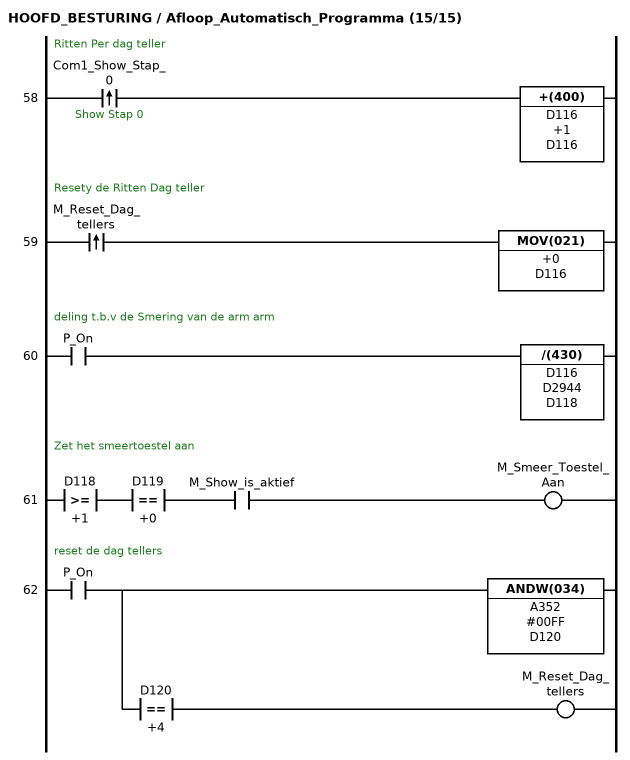
; [picture p120: HOOFD_BESTURING / Afloop_Automatisch_Programma, rungs 58-62]
; rung 58: Ritten Per dag teller
@LD Com1_Show_Stap_0  ; Show Stap 0
+(400) D116 +1 D116
; rung 59: Resety de Ritten Dag teller
@LD M_Reset_Dag_tellers
MOV(021) +0 D116
; rung 60: deling t.b.v de Smering van de arm arm
LD P_On
/(430) D116 D2944 D118
; rung 61: Zet het smeertoestel aan
LD>=S(327) D118 +1
AND=S(302) D119 +0
AND M_Show_is_aktief
OUT M_Smeer_Toestel_Aan
; rung 62: reset de dag tellers
LD P_On
ANDW(034) A352 #00FF D120
AND=S(302) D120 +4
OUT M_Reset_Dag_tellers

### Section Einde_Hoofd_Besturing
; rung 0
END(001)

## Program SIGNALEN_GROND (cyclic task 5)
Local symbols
D_FACTOR_01 D5132 REAL  ; DIVERTION FACTOR IN REAL FORMAT
D_HELP2_CNT2 D5140 REAL  ; RESULT AFTER MULIPLYING IN REAL FORMAT
D_HELP3_CNT1 D5134 REAL  ; RESULT AFTER DIVERTING IN REAL FORMAT
D_HELP3_CNT2 D5144 REAL  ; RESULT AFTER DIVERTING IN REAL FORMAT

### Section Incremental_Encoder_Decoder_1

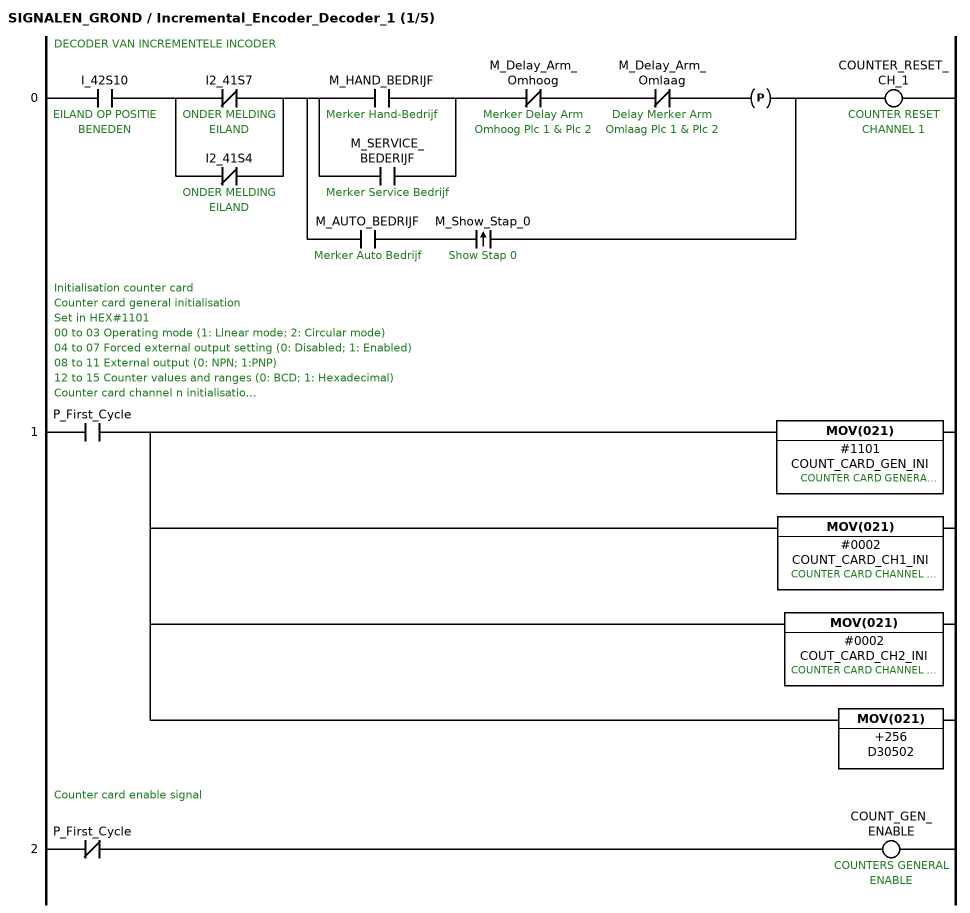
; rung 0: DECODER VAN INCREMENTELE INCODER
LD I_42S10  ; EILAND OP POSITIE BENEDEN
LDNOT I2_41S7  ; ONDER MELDING EILAND
ORNOT I2_41S4  ; ONDER MELDING EILAND
ANDLD
LD M_HAND_BEDRIJF  ; Merker Hand-Bedrijf
OR M_SERVICE_BEDERIJF  ; Merker Service Bedrijf
ANDNOT M_Delay_Arm_Omhoog  ; Merker Delay Arm Omhoog Plc 1 & Plc 2
ANDNOT M_Delay_Arm_Omlaag  ; Delay Merker Arm Omlaag Plc 1 & Plc 2
UP(521)
LD M_AUTO_BEDRIJF  ; Merker Auto Bedrijf
@AND M_Show_Stap_0  ; Show Stap 0
ORLD
ANDLD
OUT COUNTER_RESET_CH_1  ; COUNTER RESET CHANNEL 1
; rung 1: Initialisation counter card / Counter card general initialisation / Set in HEX#1101 / 00 to 03 Operating mode (1: Linear mode; 2: Circular mode) / 04 to 07 Forced external output setting (0: Disabled; 1: Enabled) / 08 to 11 External output (0: NPN; 1:PNP) / 12 to 15 Counter values and ranges (0: BCD; 1: Hexadecimal) / Counter card channel n initialisation / Set in HEX#0002 / 00 to 03 Counter 1 input types and counter reset conditions: / Input types / 0: x 1 / 1: x 2 / 2: x 4 / 3: Up and down pulses input / 4: Pulse and direction input / 04 to 07 Not used. / 08 to 15 Reset modes 00 to 11 (Mode 0 to mode 11)
LD P_First_Cycle
MOV(021) #1101 COUNT_CARD_GEN_INI  ; COUNTER CARD GENERAL INITIALISATION
MOV(021) #0002 COUNT_CARD_CH1_INI  ; COUNTER CARD CHANNEL 1 INITIALISATION
MOV(021) #0002 COUT_CARD_CH2_INI  ; COUNTER CARD CHANNEL 2 INITIALISATION
MOV(021) +256 D30502
; rung 2: Counter card enable signal
LDNOT P_First_Cycle
OUT COUNT_GEN_ENABLE  ; COUNTERS GENERAL ENABLE

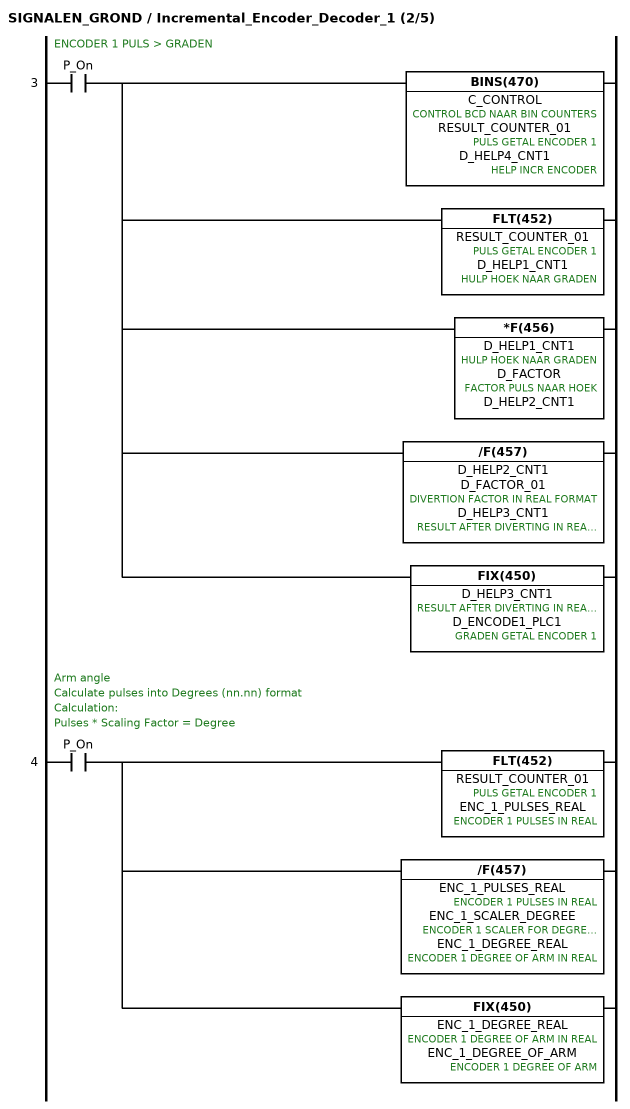
; rung 3: ENCODER 1 PULS > GRADEN
LD P_On
BINS(470) C_CONTROL RESULT_COUNTER_01 D_HELP4_CNT1  ; CONTROL BCD NAAR BIN COUNTERS, PULS GETAL ENCODER 1, HELP INCR ENCODER
FLT(452) RESULT_COUNTER_01 D_HELP1_CNT1  ; PULS GETAL ENCODER 1, HULP HOEK NAAR GRADEN
*F(456) D_HELP1_CNT1 D_FACTOR D_HELP2_CNT1  ; HULP HOEK NAAR GRADEN, FACTOR PULS NAAR HOEK
/F(457) D_HELP2_CNT1 D_FACTOR_01 D_HELP3_CNT1  ; DIVERTION FACTOR IN REAL FORMAT, RESULT AFTER DIVERTING IN REAL FORMAT
FIX(450) D_HELP3_CNT1 D_ENCODE1_PLC1  ; RESULT AFTER DIVERTING IN REAL FORMAT, GRADEN GETAL ENCODER 1
; rung 4: Arm angle / Calculate pulses into Degrees (nn.nn) format / Calculation: / Pulses * Scaling Factor = Degree
LD P_On
FLT(452) RESULT_COUNTER_01 ENC_1_PULSES_REAL  ; PULS GETAL ENCODER 1, ENCODER 1 PULSES IN REAL
/F(457) ENC_1_PULSES_REAL ENC_1_SCALER_DEGREE ENC_1_DEGREE_REAL  ; ENCODER 1 PULSES IN REAL, ENCODER 1 SCALER FOR DEGREE CALCULTION, ENCODER 1 DEGREE OF ARM IN REAL
FIX(450) ENC_1_DEGREE_REAL ENC_1_DEGREE_OF_ARM  ; ENCODER 1 DEGREE OF ARM IN REAL, ENCODER 1 DEGREE OF ARM

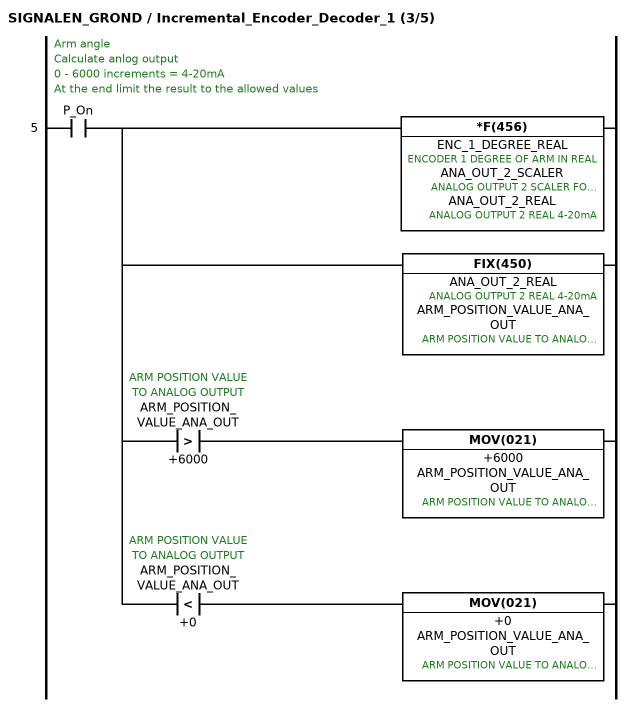
; rung 5: Arm angle / Calculate anlog output / 0 - 6000 increments = 4-20mA / At the end limit the result to the allowed values
LD P_On
OUT TR0
*F(456) ENC_1_DEGREE_REAL ANA_OUT_2_SCALER ANA_OUT_2_REAL  ; ENCODER 1 DEGREE OF ARM IN REAL, ANALOG OUTPUT 2 SCALER FOR 4-20mA, ANALOG OUTPUT 2 REAL 4-20mA
FIX(450) ANA_OUT_2_REAL ARM_POSITION_VALUE_ANA_OUT  ; ANALOG OUTPUT 2 REAL 4-20mA, ARM POSITION VALUE TO ANALOG OUTPUT
AND>S(322) ARM_POSITION_VALUE_ANA_OUT +6000  ; ARM POSITION VALUE TO ANALOG OUTPUT
MOV(021) +6000 ARM_POSITION_VALUE_ANA_OUT  ; ARM POSITION VALUE TO ANALOG OUTPUT
LD TR0
AND<S(312) ARM_POSITION_VALUE_ANA_OUT +0  ; ARM POSITION VALUE TO ANALOG OUTPUT
MOV(021) +0 ARM_POSITION_VALUE_ANA_OUT  ; ARM POSITION VALUE TO ANALOG OUTPUT

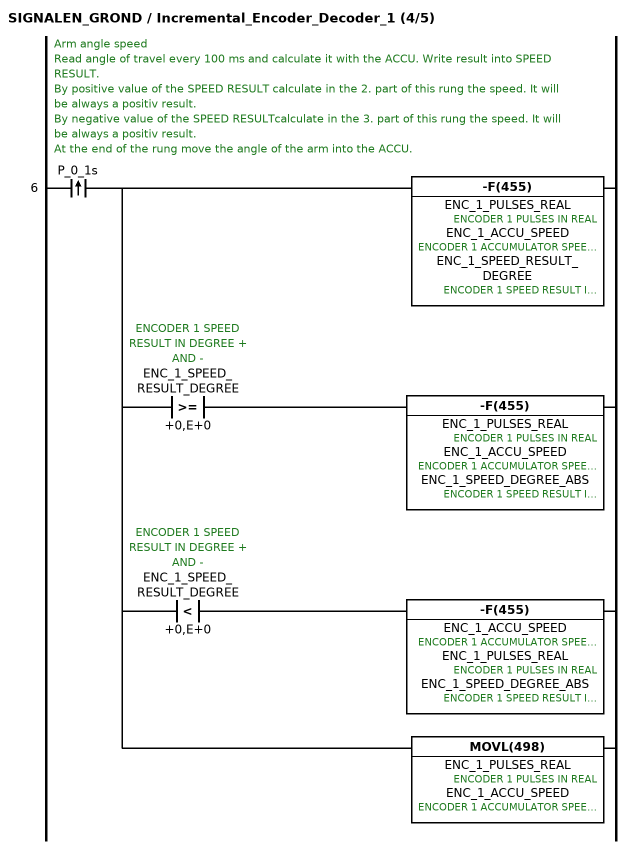
; rung 6: Arm angle speed / Read angle of travel every 100 ms and calculate it with the ACCU. Write result into SPEED RESULT. / By positive value of the SPEED RESULT calculate in the 2. part of this rung the speed. It will be always a positiv result. / By negative value of the SPEED RESULTcalculate in the 3. part of this rung the speed. It will be always a positiv result. / At the end of the rung move the angle of the arm into the ACCU.
@LD P_0_1s
OUT TR0
-F(455) ENC_1_PULSES_REAL ENC_1_ACCU_SPEED ENC_1_SPEED_RESULT_DEGREE  ; ENCODER 1 PULSES IN REAL, ENCODER 1 ACCUMULATOR SPEED CALCULATION, ENCODER 1 SPEED RESULT IN DEGREE + AND -
AND>=F(334) ENC_1_SPEED_RESULT_DEGREE +0,E+0  ; ENCODER 1 SPEED RESULT IN DEGREE + AND -
-F(455) ENC_1_PULSES_REAL ENC_1_ACCU_SPEED ENC_1_SPEED_DEGREE_ABS  ; ENCODER 1 PULSES IN REAL, ENCODER 1 ACCUMULATOR SPEED CALCULATION, ENCODER 1 SPEED RESULT IN DEGREE ABSOLUTE
LD TR0
AND<F(331) ENC_1_SPEED_RESULT_DEGREE +0,E+0  ; ENCODER 1 SPEED RESULT IN DEGREE + AND -
-F(455) ENC_1_ACCU_SPEED ENC_1_PULSES_REAL ENC_1_SPEED_DEGREE_ABS  ; ENCODER 1 ACCUMULATOR SPEED CALCULATION, ENCODER 1 PULSES IN REAL, ENCODER 1 SPEED RESULT IN DEGREE ABSOLUTE
LD TR0
MOVL(498) ENC_1_PULSES_REAL ENC_1_ACCU_SPEED  ; ENCODER 1 PULSES IN REAL, ENCODER 1 ACCUMULATOR SPEED CALCULATION

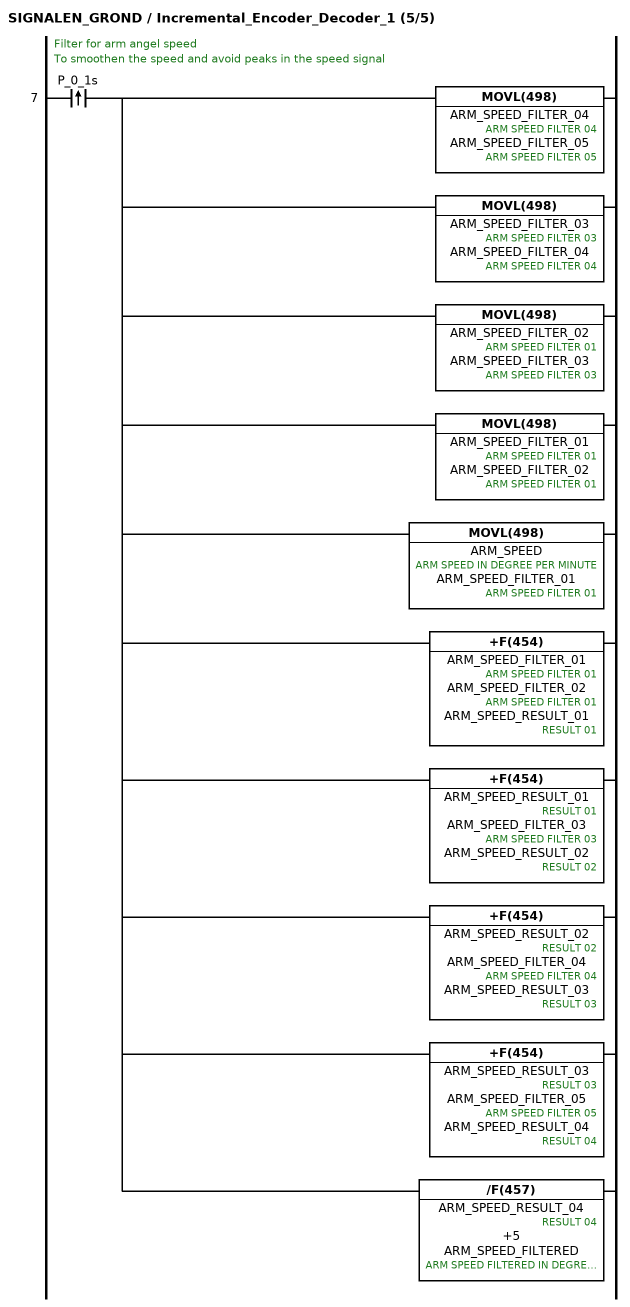
; rung 7: Filter for arm angel speed / To smoothen the speed and avoid peaks in the speed signal
@LD P_0_1s
MOVL(498) ARM_SPEED_FILTER_04 ARM_SPEED_FILTER_05  ; ARM SPEED FILTER 04, ARM SPEED FILTER 05
MOVL(498) ARM_SPEED_FILTER_03 ARM_SPEED_FILTER_04  ; ARM SPEED FILTER 03, ARM SPEED FILTER 04
MOVL(498) ARM_SPEED_FILTER_02 ARM_SPEED_FILTER_03  ; ARM SPEED FILTER 01, ARM SPEED FILTER 03
MOVL(498) ARM_SPEED_FILTER_01 ARM_SPEED_FILTER_02  ; ARM SPEED FILTER 01
MOVL(498) ARM_SPEED ARM_SPEED_FILTER_01  ; ARM SPEED IN DEGREE PER MINUTE, ARM SPEED FILTER 01
+F(454) ARM_SPEED_FILTER_01 ARM_SPEED_FILTER_02 ARM_SPEED_RESULT_01  ; ARM SPEED FILTER 01, RESULT 01
+F(454) ARM_SPEED_RESULT_01 ARM_SPEED_FILTER_03 ARM_SPEED_RESULT_02  ; RESULT 01, ARM SPEED FILTER 03, RESULT 02
+F(454) ARM_SPEED_RESULT_02 ARM_SPEED_FILTER_04 ARM_SPEED_RESULT_03  ; RESULT 02, ARM SPEED FILTER 04, RESULT 03
+F(454) ARM_SPEED_RESULT_03 ARM_SPEED_FILTER_05 ARM_SPEED_RESULT_04  ; RESULT 03, ARM SPEED FILTER 05, RESULT 04
/F(457) ARM_SPEED_RESULT_04 +5 ARM_SPEED_FILTERED  ; RESULT 04, ARM SPEED FILTERED IN DEGREE PER MINUTE

### Section Incremental_Encoder_Decoder_2

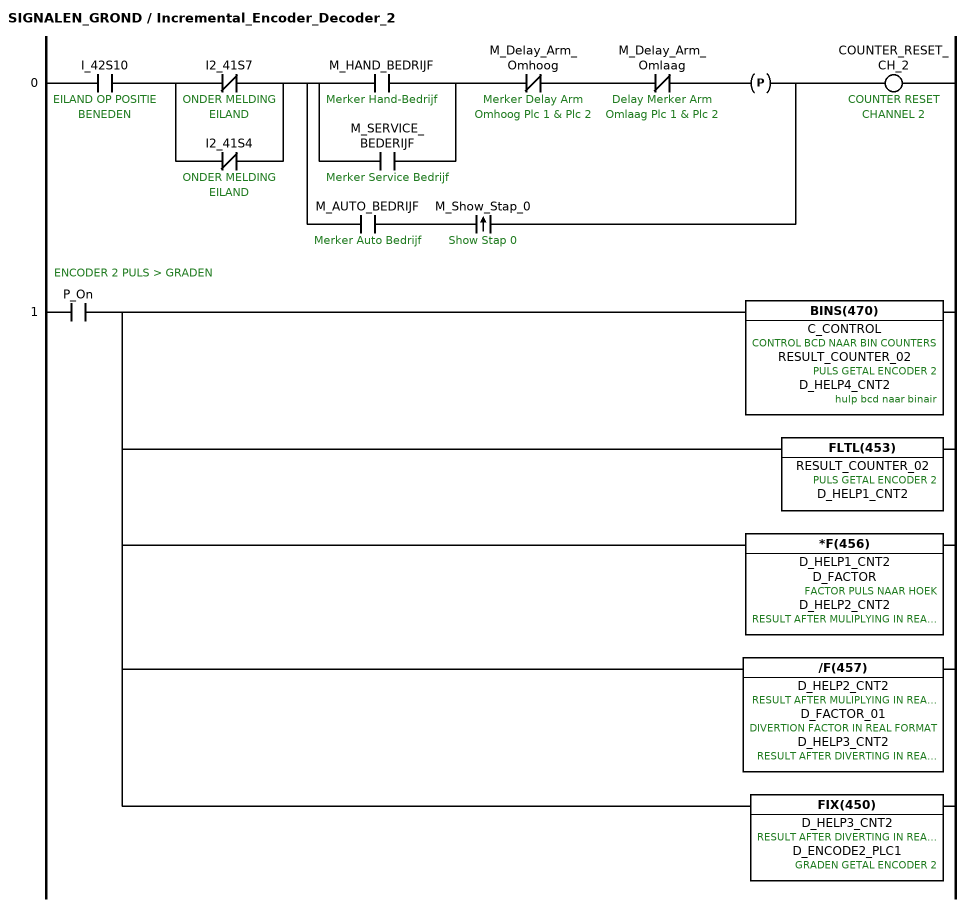
; rung 0
LD I_42S10  ; EILAND OP POSITIE BENEDEN
LDNOT I2_41S7  ; ONDER MELDING EILAND
ORNOT I2_41S4  ; ONDER MELDING EILAND
ANDLD
LD M_HAND_BEDRIJF  ; Merker Hand-Bedrijf
OR M_SERVICE_BEDERIJF  ; Merker Service Bedrijf
ANDNOT M_Delay_Arm_Omhoog  ; Merker Delay Arm Omhoog Plc 1 & Plc 2
ANDNOT M_Delay_Arm_Omlaag  ; Delay Merker Arm Omlaag Plc 1 & Plc 2
UP(521)
LD M_AUTO_BEDRIJF  ; Merker Auto Bedrijf
@AND M_Show_Stap_0  ; Show Stap 0
ORLD
ANDLD
OUT COUNTER_RESET_CH_2  ; COUNTER RESET CHANNEL 2
; rung 1: ENCODER 2 PULS > GRADEN
LD P_On
BINS(470) C_CONTROL RESULT_COUNTER_02 D_HELP4_CNT2  ; CONTROL BCD NAAR BIN COUNTERS, PULS GETAL ENCODER 2, hulp bcd naar binair
FLTL(453) RESULT_COUNTER_02 D_HELP1_CNT2  ; PULS GETAL ENCODER 2
*F(456) D_HELP1_CNT2 D_FACTOR D_HELP2_CNT2  ; FACTOR PULS NAAR HOEK, RESULT AFTER MULIPLYING IN REAL FORMAT
/F(457) D_HELP2_CNT2 D_FACTOR_01 D_HELP3_CNT2  ; RESULT AFTER MULIPLYING IN REAL FORMAT, DIVERTION FACTOR IN REAL FORMAT, RESULT AFTER DIVERTING IN REAL FORMAT
FIX(450) D_HELP3_CNT2 D_ENCODE2_PLC1  ; RESULT AFTER DIVERTING IN REAL FORMAT, GRADEN GETAL ENCODER 2

### Section Absoute_Encoder_Decoder_3

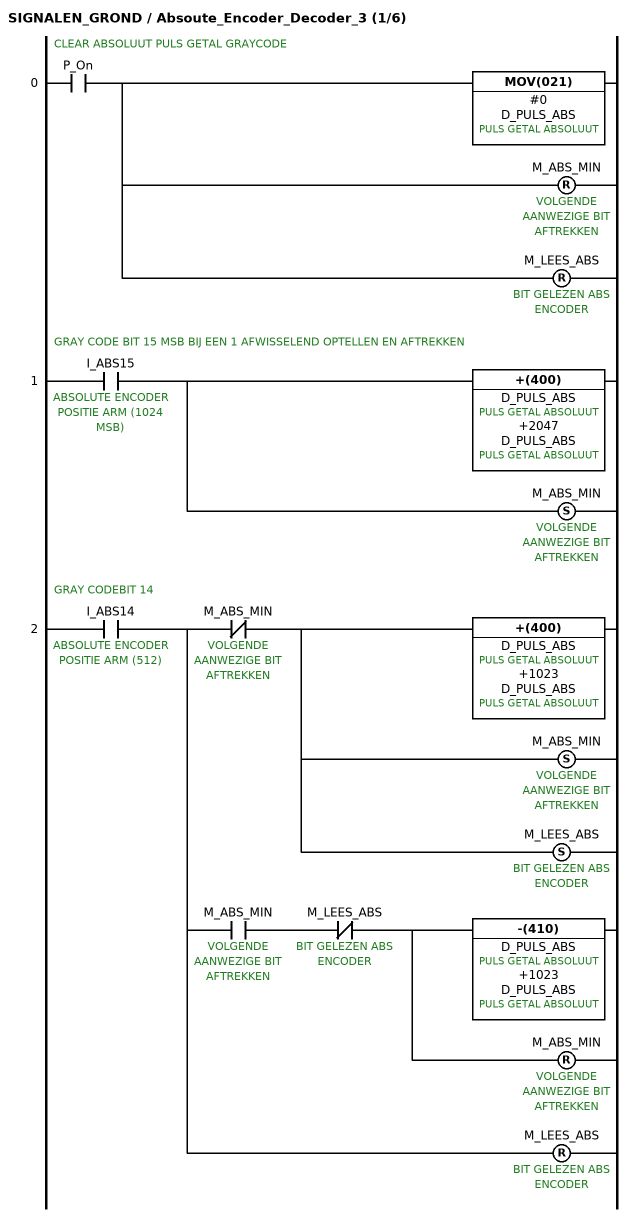
; rung 0: CLEAR ABSOLUUT PULS GETAL GRAYCODE
LD P_On
MOV(021) #0 D_PULS_ABS  ; PULS GETAL ABSOLUUT
RSET M_ABS_MIN  ; VOLGENDE  AANWEZIGE BIT AFTREKKEN
RSET M_LEES_ABS  ; BIT GELEZEN ABS ENCODER
; rung 1: GRAY CODE BIT 15 MSB BIJ EEN 1 AFWISSELEND OPTELLEN EN AFTREKKEN
LD I_ABS15  ; ABSOLUTE ENCODER POSITIE ARM (1024 MSB)
+(400) D_PULS_ABS +2047 D_PULS_ABS  ; PULS GETAL ABSOLUUT
SET M_ABS_MIN  ; VOLGENDE  AANWEZIGE BIT AFTREKKEN
; rung 2: GRAY CODEBIT 14
LD I_ABS14  ; ABSOLUTE ENCODER POSITIE ARM (512)
OUT TR0
ANDNOT M_ABS_MIN  ; VOLGENDE  AANWEZIGE BIT AFTREKKEN
+(400) D_PULS_ABS +1023 D_PULS_ABS  ; PULS GETAL ABSOLUUT
SET M_ABS_MIN  ; VOLGENDE  AANWEZIGE BIT AFTREKKEN
SET M_LEES_ABS  ; BIT GELEZEN ABS ENCODER
LD TR0
AND M_ABS_MIN  ; VOLGENDE  AANWEZIGE BIT AFTREKKEN
ANDNOT M_LEES_ABS  ; BIT GELEZEN ABS ENCODER
-(410) D_PULS_ABS +1023 D_PULS_ABS  ; PULS GETAL ABSOLUUT
RSET M_ABS_MIN  ; VOLGENDE  AANWEZIGE BIT AFTREKKEN
LD TR0
RSET M_LEES_ABS  ; BIT GELEZEN ABS ENCODER

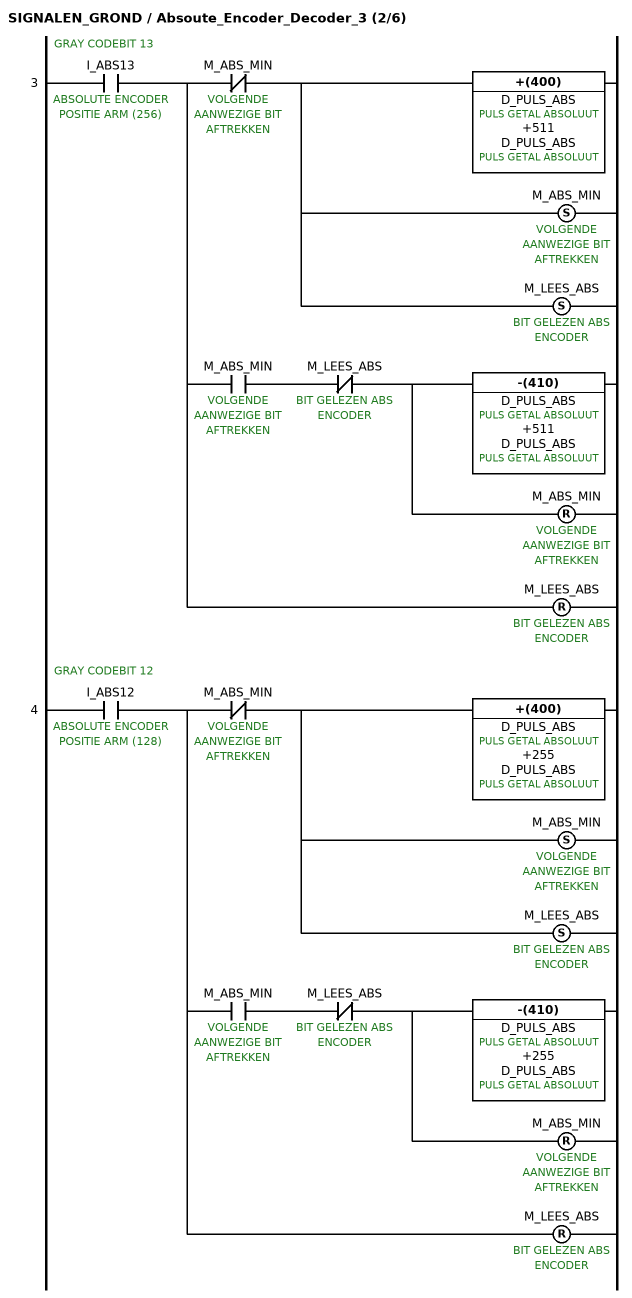
; rung 3: GRAY CODEBIT 13
LD I_ABS13  ; ABSOLUTE ENCODER POSITIE ARM (256)
OUT TR0
ANDNOT M_ABS_MIN  ; VOLGENDE  AANWEZIGE BIT AFTREKKEN
+(400) D_PULS_ABS +511 D_PULS_ABS  ; PULS GETAL ABSOLUUT
SET M_ABS_MIN  ; VOLGENDE  AANWEZIGE BIT AFTREKKEN
SET M_LEES_ABS  ; BIT GELEZEN ABS ENCODER
LD TR0
AND M_ABS_MIN  ; VOLGENDE  AANWEZIGE BIT AFTREKKEN
ANDNOT M_LEES_ABS  ; BIT GELEZEN ABS ENCODER
-(410) D_PULS_ABS +511 D_PULS_ABS  ; PULS GETAL ABSOLUUT
RSET M_ABS_MIN  ; VOLGENDE  AANWEZIGE BIT AFTREKKEN
LD TR0
RSET M_LEES_ABS  ; BIT GELEZEN ABS ENCODER
; rung 4: GRAY CODEBIT 12
LD I_ABS12  ; ABSOLUTE ENCODER POSITIE ARM (128)
OUT TR0
ANDNOT M_ABS_MIN  ; VOLGENDE  AANWEZIGE BIT AFTREKKEN
+(400) D_PULS_ABS +255 D_PULS_ABS  ; PULS GETAL ABSOLUUT
SET M_ABS_MIN  ; VOLGENDE  AANWEZIGE BIT AFTREKKEN
SET M_LEES_ABS  ; BIT GELEZEN ABS ENCODER
LD TR0
AND M_ABS_MIN  ; VOLGENDE  AANWEZIGE BIT AFTREKKEN
ANDNOT M_LEES_ABS  ; BIT GELEZEN ABS ENCODER
-(410) D_PULS_ABS +255 D_PULS_ABS  ; PULS GETAL ABSOLUUT
RSET M_ABS_MIN  ; VOLGENDE  AANWEZIGE BIT AFTREKKEN
LD TR0
RSET M_LEES_ABS  ; BIT GELEZEN ABS ENCODER

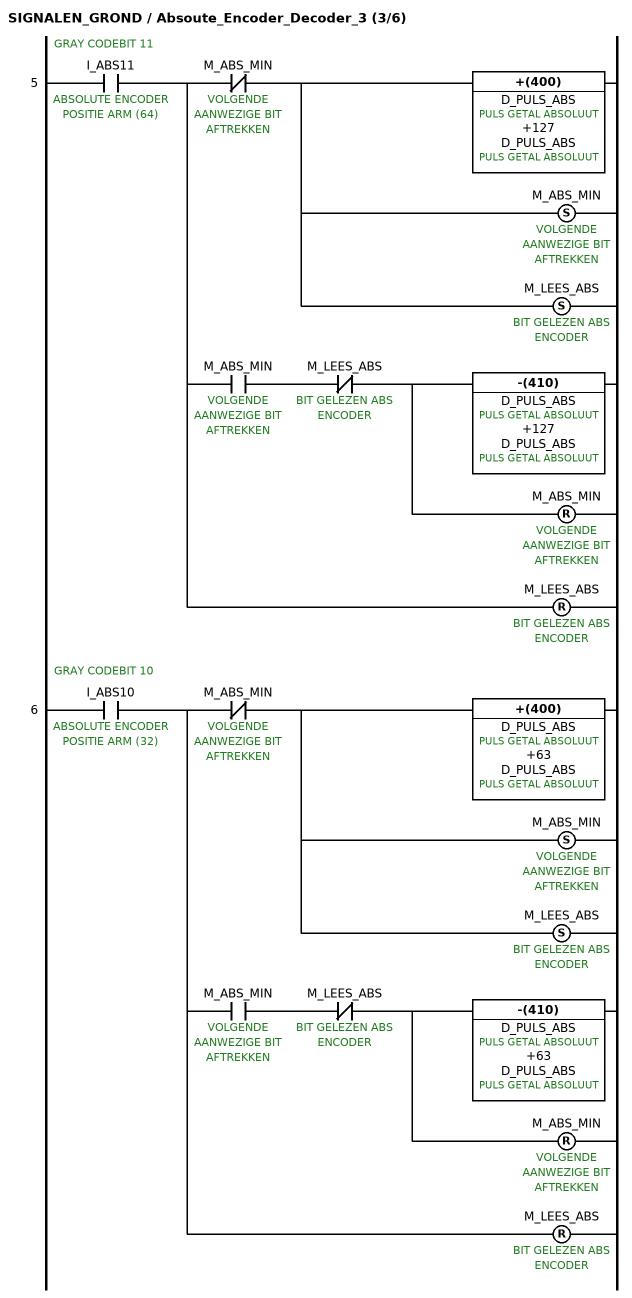
; rung 5: GRAY CODEBIT 11
LD I_ABS11  ; ABSOLUTE ENCODER POSITIE ARM (64)
OUT TR0
ANDNOT M_ABS_MIN  ; VOLGENDE  AANWEZIGE BIT AFTREKKEN
+(400) D_PULS_ABS +127 D_PULS_ABS  ; PULS GETAL ABSOLUUT
SET M_ABS_MIN  ; VOLGENDE  AANWEZIGE BIT AFTREKKEN
SET M_LEES_ABS  ; BIT GELEZEN ABS ENCODER
LD TR0
AND M_ABS_MIN  ; VOLGENDE  AANWEZIGE BIT AFTREKKEN
ANDNOT M_LEES_ABS  ; BIT GELEZEN ABS ENCODER
-(410) D_PULS_ABS +127 D_PULS_ABS  ; PULS GETAL ABSOLUUT
RSET M_ABS_MIN  ; VOLGENDE  AANWEZIGE BIT AFTREKKEN
LD TR0
RSET M_LEES_ABS  ; BIT GELEZEN ABS ENCODER
; rung 6: GRAY CODEBIT 10
LD I_ABS10  ; ABSOLUTE ENCODER POSITIE ARM (32)
OUT TR0
ANDNOT M_ABS_MIN  ; VOLGENDE  AANWEZIGE BIT AFTREKKEN
+(400) D_PULS_ABS +63 D_PULS_ABS  ; PULS GETAL ABSOLUUT
SET M_ABS_MIN  ; VOLGENDE  AANWEZIGE BIT AFTREKKEN
SET M_LEES_ABS  ; BIT GELEZEN ABS ENCODER
LD TR0
AND M_ABS_MIN  ; VOLGENDE  AANWEZIGE BIT AFTREKKEN
ANDNOT M_LEES_ABS  ; BIT GELEZEN ABS ENCODER
-(410) D_PULS_ABS +63 D_PULS_ABS  ; PULS GETAL ABSOLUUT
RSET M_ABS_MIN  ; VOLGENDE  AANWEZIGE BIT AFTREKKEN
LD TR0
RSET M_LEES_ABS  ; BIT GELEZEN ABS ENCODER

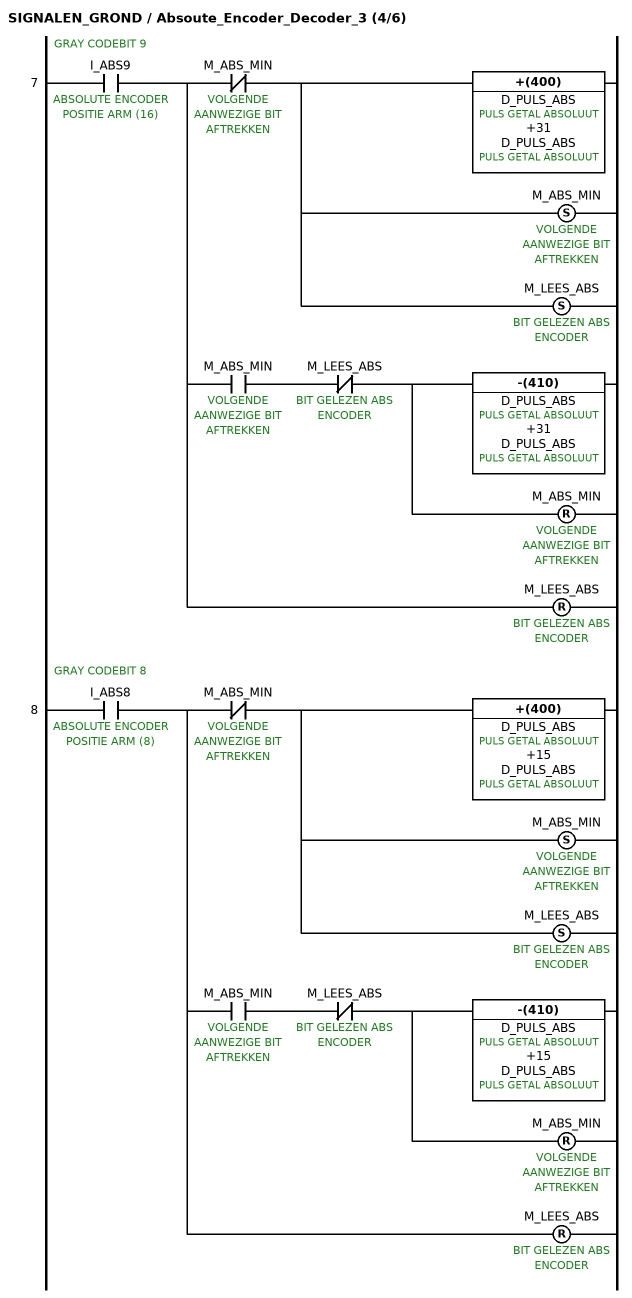
; rung 7: GRAY CODEBIT 9
LD I_ABS9  ; ABSOLUTE ENCODER POSITIE ARM (16)
OUT TR0
ANDNOT M_ABS_MIN  ; VOLGENDE  AANWEZIGE BIT AFTREKKEN
+(400) D_PULS_ABS +31 D_PULS_ABS  ; PULS GETAL ABSOLUUT
SET M_ABS_MIN  ; VOLGENDE  AANWEZIGE BIT AFTREKKEN
SET M_LEES_ABS  ; BIT GELEZEN ABS ENCODER
LD TR0
AND M_ABS_MIN  ; VOLGENDE  AANWEZIGE BIT AFTREKKEN
ANDNOT M_LEES_ABS  ; BIT GELEZEN ABS ENCODER
-(410) D_PULS_ABS +31 D_PULS_ABS  ; PULS GETAL ABSOLUUT
RSET M_ABS_MIN  ; VOLGENDE  AANWEZIGE BIT AFTREKKEN
LD TR0
RSET M_LEES_ABS  ; BIT GELEZEN ABS ENCODER
; rung 8: GRAY CODEBIT 8
LD I_ABS8  ; ABSOLUTE ENCODER POSITIE ARM (8)
OUT TR0
ANDNOT M_ABS_MIN  ; VOLGENDE  AANWEZIGE BIT AFTREKKEN
+(400) D_PULS_ABS +15 D_PULS_ABS  ; PULS GETAL ABSOLUUT
SET M_ABS_MIN  ; VOLGENDE  AANWEZIGE BIT AFTREKKEN
SET M_LEES_ABS  ; BIT GELEZEN ABS ENCODER
LD TR0
AND M_ABS_MIN  ; VOLGENDE  AANWEZIGE BIT AFTREKKEN
ANDNOT M_LEES_ABS  ; BIT GELEZEN ABS ENCODER
-(410) D_PULS_ABS +15 D_PULS_ABS  ; PULS GETAL ABSOLUUT
RSET M_ABS_MIN  ; VOLGENDE  AANWEZIGE BIT AFTREKKEN
LD TR0
RSET M_LEES_ABS  ; BIT GELEZEN ABS ENCODER

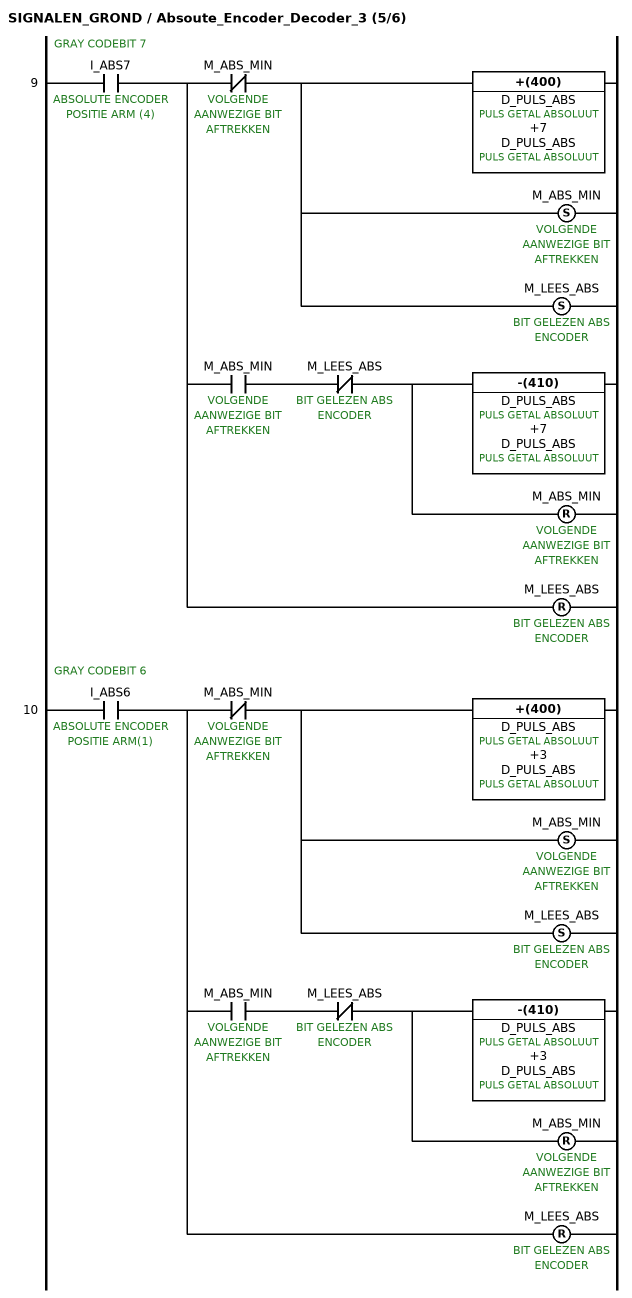
; rung 9: GRAY CODEBIT 7
LD I_ABS7  ; ABSOLUTE ENCODER POSITIE ARM (4)
OUT TR0
ANDNOT M_ABS_MIN  ; VOLGENDE  AANWEZIGE BIT AFTREKKEN
+(400) D_PULS_ABS +7 D_PULS_ABS  ; PULS GETAL ABSOLUUT
SET M_ABS_MIN  ; VOLGENDE  AANWEZIGE BIT AFTREKKEN
SET M_LEES_ABS  ; BIT GELEZEN ABS ENCODER
LD TR0
AND M_ABS_MIN  ; VOLGENDE  AANWEZIGE BIT AFTREKKEN
ANDNOT M_LEES_ABS  ; BIT GELEZEN ABS ENCODER
-(410) D_PULS_ABS +7 D_PULS_ABS  ; PULS GETAL ABSOLUUT
RSET M_ABS_MIN  ; VOLGENDE  AANWEZIGE BIT AFTREKKEN
LD TR0
RSET M_LEES_ABS  ; BIT GELEZEN ABS ENCODER
; rung 10: GRAY CODEBIT 6
LD I_ABS6  ; ABSOLUTE ENCODER POSITIE ARM(1)
OUT TR0
ANDNOT M_ABS_MIN  ; VOLGENDE  AANWEZIGE BIT AFTREKKEN
+(400) D_PULS_ABS +3 D_PULS_ABS  ; PULS GETAL ABSOLUUT
SET M_ABS_MIN  ; VOLGENDE  AANWEZIGE BIT AFTREKKEN
SET M_LEES_ABS  ; BIT GELEZEN ABS ENCODER
LD TR0
AND M_ABS_MIN  ; VOLGENDE  AANWEZIGE BIT AFTREKKEN
ANDNOT M_LEES_ABS  ; BIT GELEZEN ABS ENCODER
-(410) D_PULS_ABS +3 D_PULS_ABS  ; PULS GETAL ABSOLUUT
RSET M_ABS_MIN  ; VOLGENDE  AANWEZIGE BIT AFTREKKEN
LD TR0
RSET M_LEES_ABS  ; BIT GELEZEN ABS ENCODER

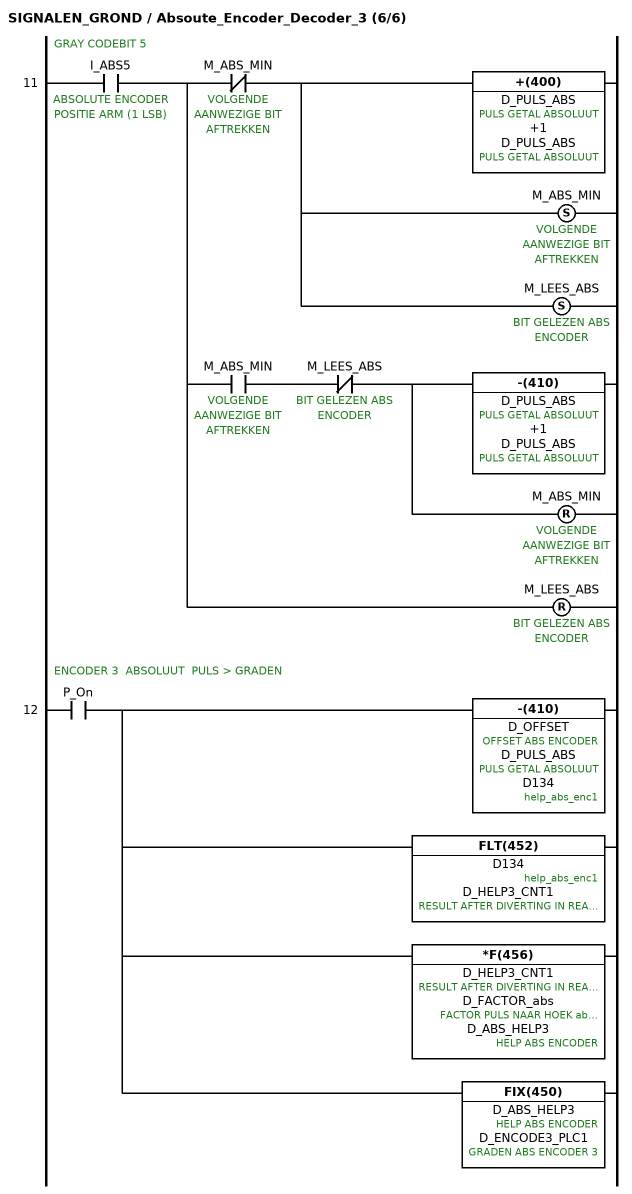
; rung 11: GRAY CODEBIT 5
LD I_ABS5  ; ABSOLUTE ENCODER POSITIE ARM (1 LSB)
OUT TR0
ANDNOT M_ABS_MIN  ; VOLGENDE  AANWEZIGE BIT AFTREKKEN
+(400) D_PULS_ABS +1 D_PULS_ABS  ; PULS GETAL ABSOLUUT
SET M_ABS_MIN  ; VOLGENDE  AANWEZIGE BIT AFTREKKEN
SET M_LEES_ABS  ; BIT GELEZEN ABS ENCODER
LD TR0
AND M_ABS_MIN  ; VOLGENDE  AANWEZIGE BIT AFTREKKEN
ANDNOT M_LEES_ABS  ; BIT GELEZEN ABS ENCODER
-(410) D_PULS_ABS +1 D_PULS_ABS  ; PULS GETAL ABSOLUUT
RSET M_ABS_MIN  ; VOLGENDE  AANWEZIGE BIT AFTREKKEN
LD TR0
RSET M_LEES_ABS  ; BIT GELEZEN ABS ENCODER
; rung 12: ENCODER 3  ABSOLUUT  PULS > GRADEN
LD P_On
-(410) D_OFFSET D_PULS_ABS D134  ; OFFSET ABS ENCODER, PULS GETAL ABSOLUUT, help_abs_enc1
FLT(452) D134 D_HELP3_CNT1  ; help_abs_enc1, RESULT AFTER DIVERTING IN REAL FORMAT
*F(456) D_HELP3_CNT1 D_FACTOR_abs D_ABS_HELP3  ; RESULT AFTER DIVERTING IN REAL FORMAT, FACTOR PULS NAAR HOEK abs encoder, HELP ABS ENCODER
FIX(450) D_ABS_HELP3 D_ENCODE3_PLC1  ; HELP ABS ENCODER, GRADEN ABS ENCODER 3

### Section Controle_Positie_Arm

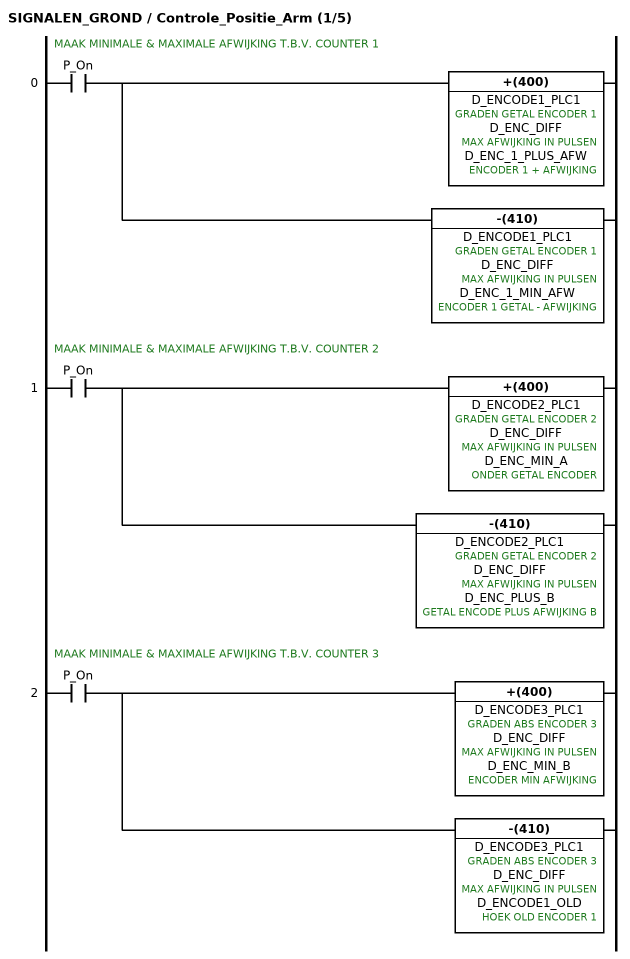
; rung 0: MAAK MINIMALE & MAXIMALE AFWIJKING T.B.V. COUNTER 1
LD P_On
+(400) D_ENCODE1_PLC1 D_ENC_DIFF D_ENC_1_PLUS_AFW  ; GRADEN GETAL ENCODER 1, MAX AFWIJKING IN PULSEN, ENCODER 1 + AFWIJKING
-(410) D_ENCODE1_PLC1 D_ENC_DIFF D_ENC_1_MIN_AFW  ; GRADEN GETAL ENCODER 1, MAX AFWIJKING IN PULSEN, ENCODER 1 GETAL - AFWIJKING
; rung 1: MAAK MINIMALE & MAXIMALE AFWIJKING T.B.V. COUNTER 2
LD P_On
+(400) D_ENCODE2_PLC1 D_ENC_DIFF D_ENC_MIN_A  ; GRADEN GETAL ENCODER 2, MAX AFWIJKING IN PULSEN, ONDER GETAL ENCODER
-(410) D_ENCODE2_PLC1 D_ENC_DIFF D_ENC_PLUS_B  ; GRADEN GETAL ENCODER 2, MAX AFWIJKING IN PULSEN, GETAL ENCODE PLUS AFWIJKING B
; rung 2: MAAK MINIMALE & MAXIMALE AFWIJKING T.B.V. COUNTER 3
LD P_On
+(400) D_ENCODE3_PLC1 D_ENC_DIFF D_ENC_MIN_B  ; GRADEN ABS ENCODER 3, MAX AFWIJKING IN PULSEN, ENCODER MIN AFWIJKING
-(410) D_ENCODE3_PLC1 D_ENC_DIFF D_ENCODE1_OLD  ; GRADEN ABS ENCODER 3, MAX AFWIJKING IN PULSEN, HOEK OLD ENCODER 1

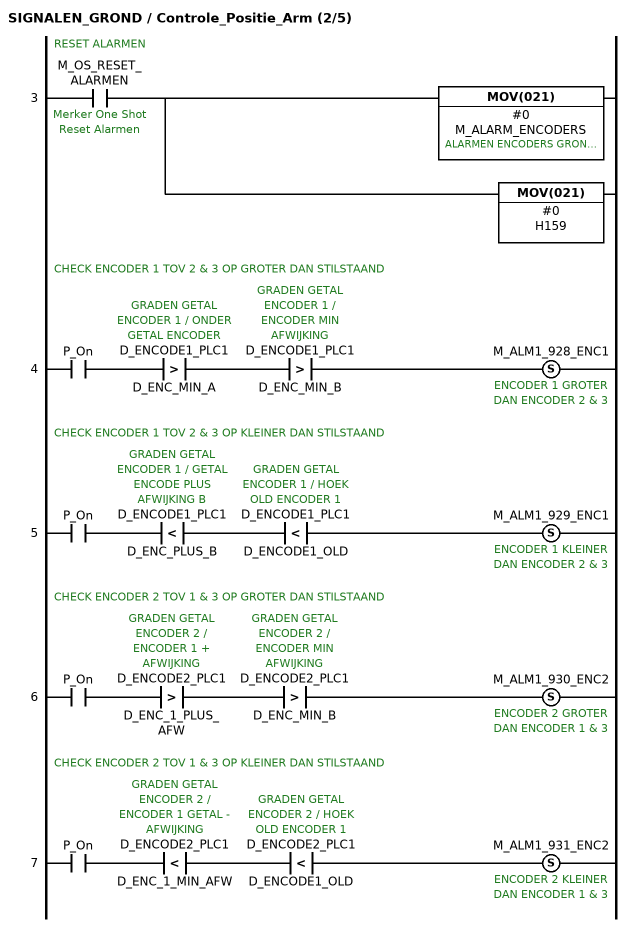
; rung 3: RESET ALARMEN
LD M_OS_RESET_ALARMEN  ; Merker One Shot Reset Alarmen
MOV(021) #0 M_ALARM_ENCODERS  ; ALARMEN ENCODERS GROND 928-943
MOV(021) #0 H159
; rung 4: CHECK ENCODER 1 TOV 2 & 3 OP GROTER DAN STILSTAAND
LD P_On
AND>S(322) D_ENCODE1_PLC1 D_ENC_MIN_A  ; GRADEN GETAL ENCODER 1, ONDER GETAL ENCODER
AND>S(322) D_ENCODE1_PLC1 D_ENC_MIN_B  ; GRADEN GETAL ENCODER 1, ENCODER MIN AFWIJKING
SET M_ALM1_928_ENC1  ; ENCODER 1 GROTER DAN ENCODER 2 & 3
; rung 5: CHECK ENCODER 1 TOV 2 & 3 OP KLEINER DAN STILSTAAND
LD P_On
AND<S(312) D_ENCODE1_PLC1 D_ENC_PLUS_B  ; GRADEN GETAL ENCODER 1, GETAL ENCODE PLUS AFWIJKING B
AND<S(312) D_ENCODE1_PLC1 D_ENCODE1_OLD  ; GRADEN GETAL ENCODER 1, HOEK OLD ENCODER 1
SET M_ALM1_929_ENC1  ; ENCODER 1 KLEINER DAN ENCODER 2 & 3
; rung 6: CHECK ENCODER 2 TOV 1 & 3 OP GROTER DAN STILSTAAND
LD P_On
AND>S(322) D_ENCODE2_PLC1 D_ENC_1_PLUS_AFW  ; GRADEN GETAL ENCODER 2, ENCODER 1 + AFWIJKING
AND>S(322) D_ENCODE2_PLC1 D_ENC_MIN_B  ; GRADEN GETAL ENCODER 2, ENCODER MIN AFWIJKING
SET M_ALM1_930_ENC2  ; ENCODER 2 GROTER DAN ENCODER 1 & 3
; rung 7: CHECK ENCODER 2 TOV 1 & 3 OP KLEINER DAN STILSTAAND
LD P_On
AND<S(312) D_ENCODE2_PLC1 D_ENC_1_MIN_AFW  ; GRADEN GETAL ENCODER 2, ENCODER 1 GETAL - AFWIJKING
AND<S(312) D_ENCODE2_PLC1 D_ENCODE1_OLD  ; GRADEN GETAL ENCODER 2, HOEK OLD ENCODER 1
SET M_ALM1_931_ENC2  ; ENCODER 2 KLEINER DAN ENCODER 1 & 3

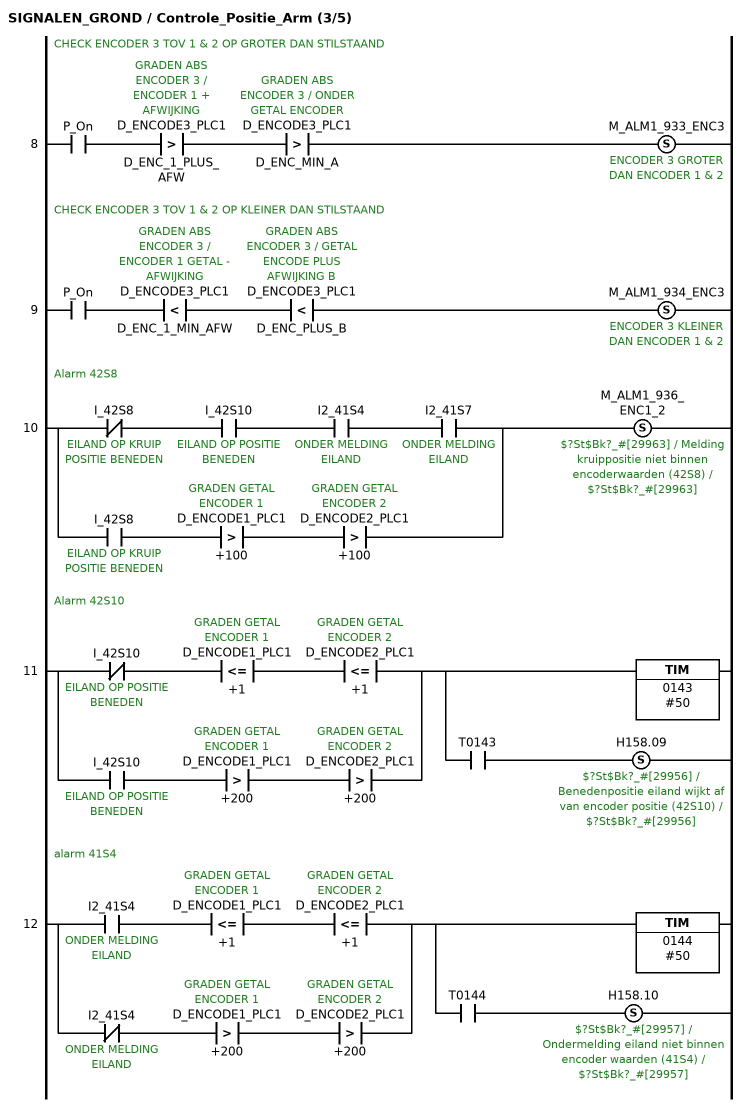
; rung 8: CHECK ENCODER 3 TOV 1 & 2 OP GROTER DAN STILSTAAND
LD P_On
AND>S(322) D_ENCODE3_PLC1 D_ENC_1_PLUS_AFW  ; GRADEN ABS ENCODER 3, ENCODER 1 + AFWIJKING
AND>S(322) D_ENCODE3_PLC1 D_ENC_MIN_A  ; GRADEN ABS ENCODER 3, ONDER GETAL ENCODER
SET M_ALM1_933_ENC3  ; ENCODER 3 GROTER DAN ENCODER 1 & 2
; rung 9: CHECK ENCODER 3 TOV 1 & 2 OP KLEINER DAN STILSTAAND
LD P_On
AND<S(312) D_ENCODE3_PLC1 D_ENC_1_MIN_AFW  ; GRADEN ABS ENCODER 3, ENCODER 1 GETAL - AFWIJKING
AND<S(312) D_ENCODE3_PLC1 D_ENC_PLUS_B  ; GRADEN ABS ENCODER 3, GETAL ENCODE PLUS AFWIJKING B
SET M_ALM1_934_ENC3  ; ENCODER 3 KLEINER DAN ENCODER 1 & 2
; rung 10: Alarm 42S8
LDNOT I_42S8  ; EILAND OP KRUIP POSITIE BENEDEN
AND I_42S10  ; EILAND OP POSITIE BENEDEN
AND I2_41S4  ; ONDER MELDING EILAND
AND I2_41S7  ; ONDER MELDING EILAND
LD I_42S8  ; EILAND OP KRUIP POSITIE BENEDEN
AND>S(322) D_ENCODE1_PLC1 +100  ; GRADEN GETAL ENCODER 1
AND>S(322) D_ENCODE2_PLC1 +100  ; GRADEN GETAL ENCODER 2
ORLD
SET M_ALM1_936_ENC1_2  ; $?St$Bk?_#[29963] / Melding kruippositie niet binnen encoderwaarden (42S8) / $?St$Bk?_#[29963]
; rung 11: Alarm 42S10
LDNOT I_42S10  ; EILAND OP POSITIE BENEDEN
AND<=S(317) D_ENCODE1_PLC1 +1  ; GRADEN GETAL ENCODER 1
AND<=S(317) D_ENCODE2_PLC1 +1  ; GRADEN GETAL ENCODER 2
LD I_42S10  ; EILAND OP POSITIE BENEDEN
AND>S(322) D_ENCODE1_PLC1 +200  ; GRADEN GETAL ENCODER 1
AND>S(322) D_ENCODE2_PLC1 +200  ; GRADEN GETAL ENCODER 2
ORLD
TIM 0143 #50
AND T0143
SET H158.09  ; $?St$Bk?_#[29956] / Benedenpositie eiland wijkt af van encoder positie (42S10) / $?St$Bk?_#[29956]
; rung 12: alarm 41S4
LD I2_41S4  ; ONDER MELDING EILAND
AND<=S(317) D_ENCODE1_PLC1 +1  ; GRADEN GETAL ENCODER 1
AND<=S(317) D_ENCODE2_PLC1 +1  ; GRADEN GETAL ENCODER 2
LDNOT I2_41S4  ; ONDER MELDING EILAND
AND>S(322) D_ENCODE1_PLC1 +200  ; GRADEN GETAL ENCODER 1
AND>S(322) D_ENCODE2_PLC1 +200  ; GRADEN GETAL ENCODER 2
ORLD
TIM 0144 #50
AND T0144
SET H158.10  ; $?St$Bk?_#[29957] / Ondermelding eiland niet binnen encoder waarden (41S4) / $?St$Bk?_#[29957]

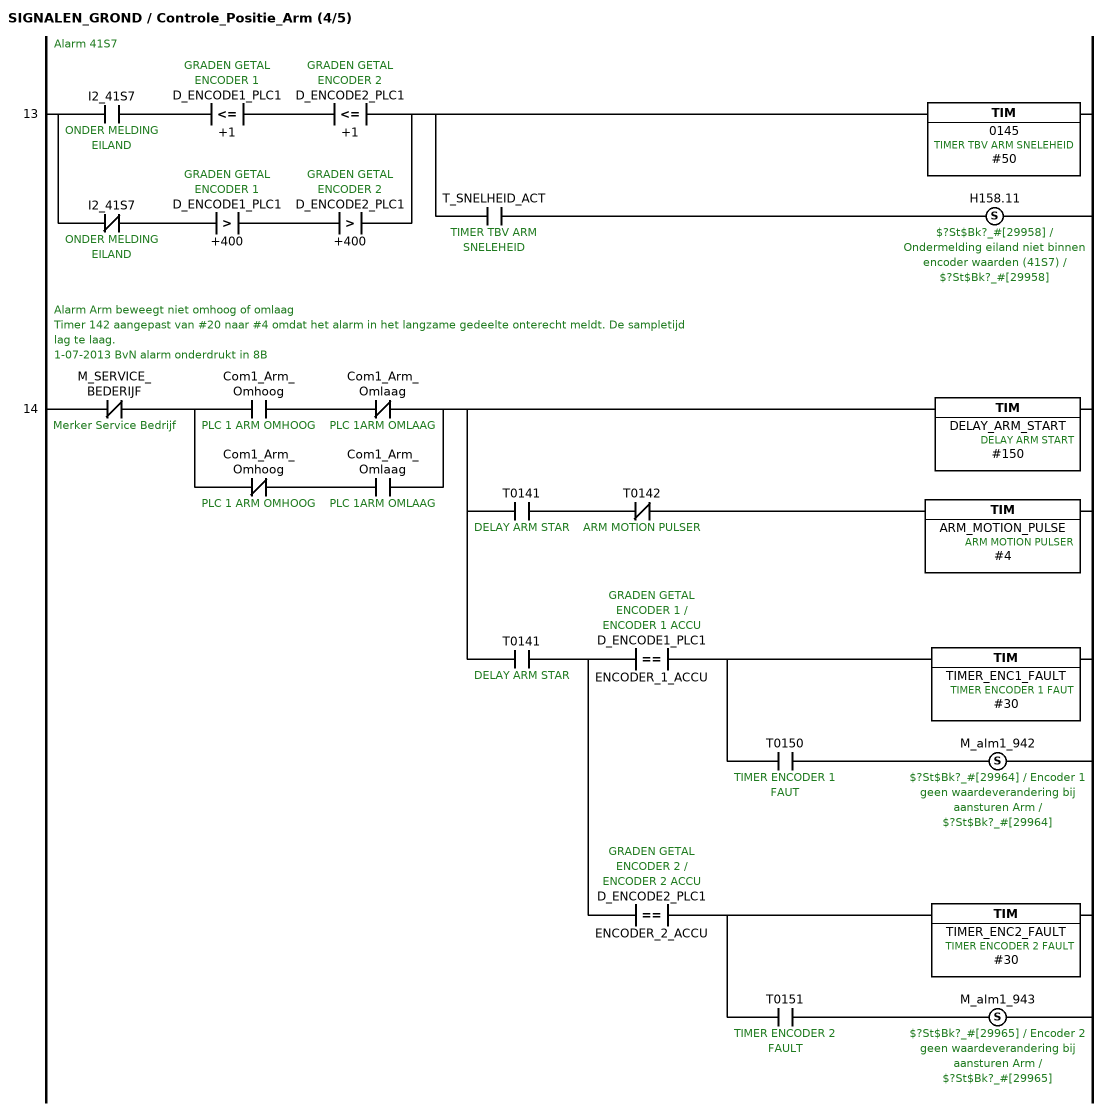
; rung 13: Alarm 41S7
LD I2_41S7  ; ONDER MELDING EILAND
AND<=S(317) D_ENCODE1_PLC1 +1  ; GRADEN GETAL ENCODER 1
AND<=S(317) D_ENCODE2_PLC1 +1  ; GRADEN GETAL ENCODER 2
LDNOT I2_41S7  ; ONDER MELDING EILAND
AND>S(322) D_ENCODE1_PLC1 +400  ; GRADEN GETAL ENCODER 1
AND>S(322) D_ENCODE2_PLC1 +400  ; GRADEN GETAL ENCODER 2
ORLD
TIM 0145 #50  ; TIMER TBV ARM SNELEHEID
AND T_SNELHEID_ACT  ; TIMER TBV ARM SNELEHEID
SET H158.11  ; $?St$Bk?_#[29958] / Ondermelding eiland niet binnen encoder waarden (41S7) / $?St$Bk?_#[29958]
; rung 14: Alarm Arm beweegt niet omhoog of omlaag / Timer 142 aangepast van #20 naar #4 omdat het alarm in het langzame gedeelte onterecht meldt. De sampletijd / lag te laag. / 1-07-2013 BvN alarm onderdrukt in 8B
LDNOT M_SERVICE_BEDERIJF  ; Merker Service Bedrijf
LD Com1_Arm_Omhoog  ; PLC 1 ARM OMHOOG
ANDNOT Com1_Arm_Omlaag  ; PLC 1ARM OMLAAG
LDNOT Com1_Arm_Omhoog  ; PLC 1 ARM OMHOOG
AND Com1_Arm_Omlaag  ; PLC 1ARM OMLAAG
ORLD
ANDLD
OUT TR0
TIM DELAY_ARM_START #150  ; DELAY ARM START
AND T0141  ; DELAY ARM STAR
ANDNOT T0142  ; ARM MOTION PULSER
TIM ARM_MOTION_PULSE #4  ; ARM MOTION PULSER
LD TR0
AND T0141  ; DELAY ARM STAR
OUT TR0
AND=(300) D_ENCODE1_PLC1 ENCODER_1_ACCU  ; GRADEN GETAL ENCODER 1, ENCODER 1 ACCU
TIM TIMER_ENC1_FAULT #30  ; TIMER ENCODER 1 FAUT
AND T0150  ; TIMER ENCODER 1 FAUT
SET M_alm1_942  ; $?St$Bk?_#[29964] / Encoder 1 geen waardeverandering bij aansturen Arm / $?St$Bk?_#[29964]
LD TR0
AND=(300) D_ENCODE2_PLC1 ENCODER_2_ACCU  ; GRADEN GETAL ENCODER 2, ENCODER 2 ACCU
TIM TIMER_ENC2_FAULT #30  ; TIMER ENCODER 2 FAULT
AND T0151  ; TIMER ENCODER 2 FAULT
SET M_alm1_943  ; $?St$Bk?_#[29965] / Encoder 2 geen waardeverandering bij aansturen Arm / $?St$Bk?_#[29965]

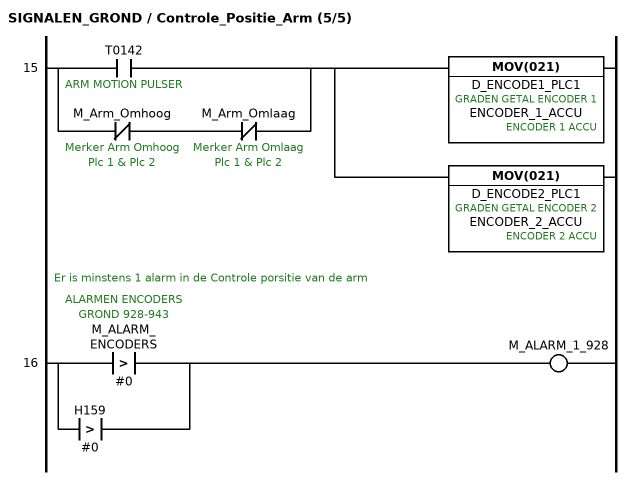
; rung 15
LD T0142  ; ARM MOTION PULSER
LDNOT M_Arm_Omhoog  ; Merker Arm Omhoog Plc 1 & Plc 2
ANDNOT M_Arm_Omlaag  ; Merker Arm Omlaag Plc 1 & Plc 2
ORLD
MOV(021) D_ENCODE1_PLC1 ENCODER_1_ACCU  ; GRADEN GETAL ENCODER 1, ENCODER 1 ACCU
MOV(021) D_ENCODE2_PLC1 ENCODER_2_ACCU  ; GRADEN GETAL ENCODER 2, ENCODER 2 ACCU
; rung 16: Er is minstens 1 alarm in de Controle porsitie van de arm
LD>(320) M_ALARM_ENCODERS #0  ; ALARMEN ENCODERS GROND 928-943
OR>(320) H159 #0
OUT M_ALARM_1_928

### Section Controle_Snelheid_Arm

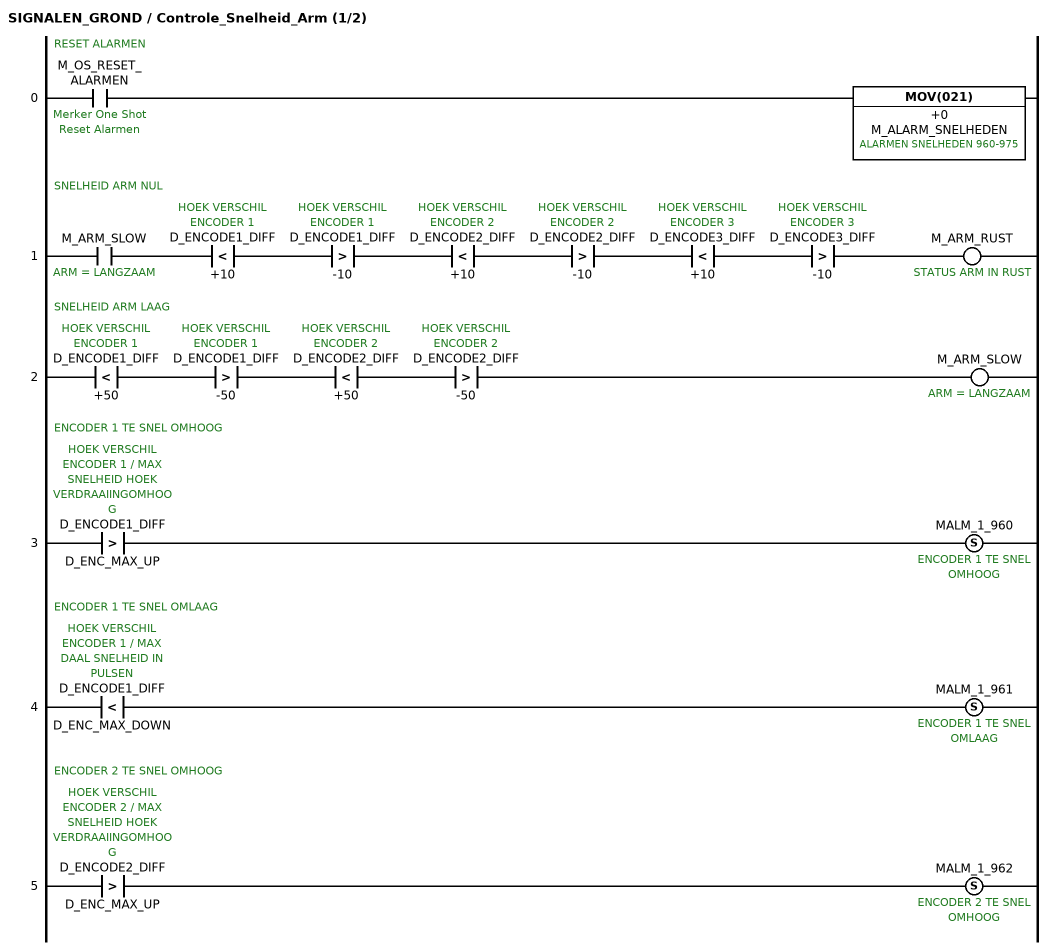
; rung 0: RESET ALARMEN
LD M_OS_RESET_ALARMEN  ; Merker One Shot Reset Alarmen
MOV(021) +0 M_ALARM_SNELHEDEN  ; ALARMEN SNELHEDEN 960-975
; rung 1: SNELHEID ARM NUL
LD M_ARM_SLOW  ; ARM = LANGZAAM
AND<S(312) D_ENCODE1_DIFF +10  ; HOEK VERSCHIL ENCODER 1
AND>S(322) D_ENCODE1_DIFF -10  ; HOEK VERSCHIL ENCODER 1
AND<S(312) D_ENCODE2_DIFF +10  ; HOEK VERSCHIL ENCODER 2
AND>S(322) D_ENCODE2_DIFF -10  ; HOEK VERSCHIL ENCODER 2
AND<S(312) D_ENCODE3_DIFF +10  ; HOEK VERSCHIL ENCODER 3
AND>S(322) D_ENCODE3_DIFF -10  ; HOEK VERSCHIL ENCODER 3
OUT M_ARM_RUST  ; STATUS ARM IN RUST
; rung 2: SNELHEID ARM LAAG
LD<S(312) D_ENCODE1_DIFF +50  ; HOEK VERSCHIL ENCODER 1
AND>S(322) D_ENCODE1_DIFF -50  ; HOEK VERSCHIL ENCODER 1
AND<S(312) D_ENCODE2_DIFF +50  ; HOEK VERSCHIL ENCODER 2
AND>S(322) D_ENCODE2_DIFF -50  ; HOEK VERSCHIL ENCODER 2
OUT M_ARM_SLOW  ; ARM = LANGZAAM
; rung 3: ENCODER 1 TE SNEL OMHOOG
LD>S(322) D_ENCODE1_DIFF D_ENC_MAX_UP  ; HOEK VERSCHIL ENCODER 1, MAX SNELHEID HOEK VERDRAAIINGOMHOOG
SET MALM_1_960  ; ENCODER 1 TE SNEL OMHOOG
; rung 4: ENCODER 1 TE SNEL OMLAAG
LD<S(312) D_ENCODE1_DIFF D_ENC_MAX_DOWN  ; HOEK VERSCHIL ENCODER 1, MAX DAAL SNELHEID IN PULSEN
SET MALM_1_961  ; ENCODER 1 TE SNEL OMLAAG
; rung 5: ENCODER 2 TE SNEL OMHOOG
LD>S(322) D_ENCODE2_DIFF D_ENC_MAX_UP  ; HOEK VERSCHIL ENCODER 2, MAX SNELHEID HOEK VERDRAAIINGOMHOOG
SET MALM_1_962  ; ENCODER 2 TE SNEL OMHOOG

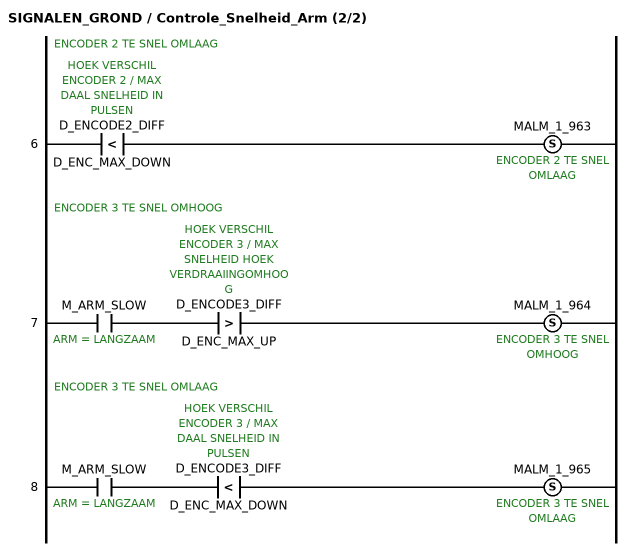
; rung 6: ENCODER 2 TE SNEL OMLAAG
LD<S(312) D_ENCODE2_DIFF D_ENC_MAX_DOWN  ; HOEK VERSCHIL ENCODER 2, MAX DAAL SNELHEID IN PULSEN
SET MALM_1_963  ; ENCODER 2 TE SNEL OMLAAG
; rung 7: ENCODER 3 TE SNEL OMHOOG
LD M_ARM_SLOW  ; ARM = LANGZAAM
AND>S(322) D_ENCODE3_DIFF D_ENC_MAX_UP  ; HOEK VERSCHIL ENCODER 3, MAX SNELHEID HOEK VERDRAAIINGOMHOOG
SET MALM_1_964  ; ENCODER 3 TE SNEL OMHOOG
; rung 8: ENCODER 3 TE SNEL OMLAAG
LD M_ARM_SLOW  ; ARM = LANGZAAM
AND<S(312) D_ENCODE3_DIFF D_ENC_MAX_DOWN  ; HOEK VERSCHIL ENCODER 3, MAX DAAL SNELHEID IN PULSEN
SET MALM_1_965  ; ENCODER 3 TE SNEL OMLAAG

### Section Einde_Signalen_Grond
; rung 0
END(001)

## Program BESTURING_GROND (cyclic task 6)
Local symbols
M_Reset_Dag_tellers W116.14 BOOL

### Section Tourniquets

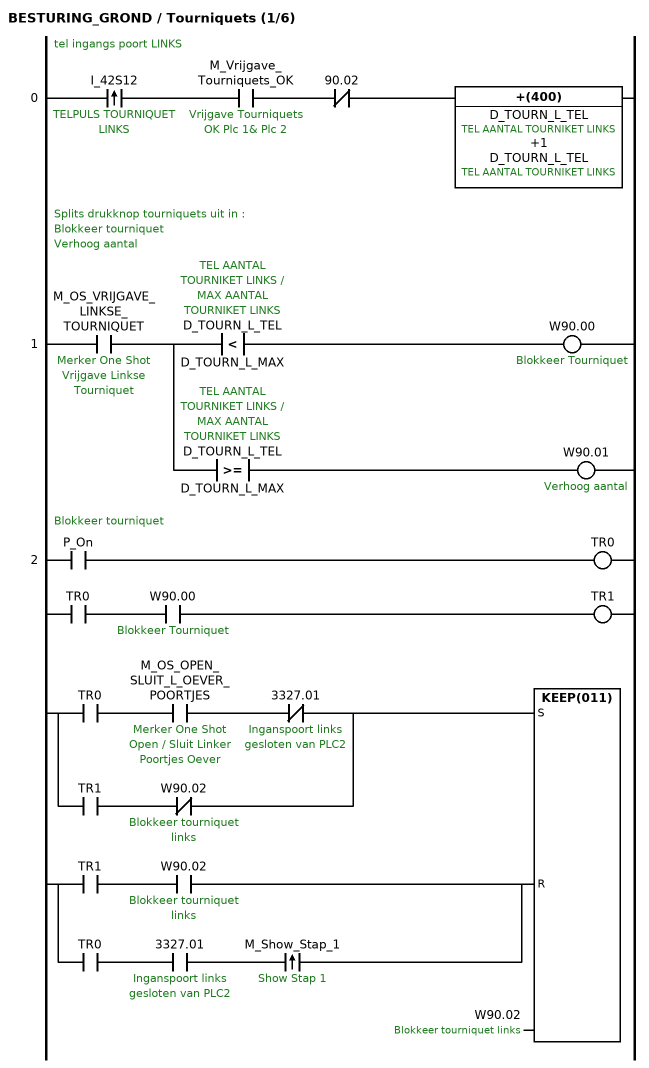
; rung 0: tel ingangs poort LINKS
@LD I_42S12  ; TELPULS TOURNIQUET LINKS
AND M_Vrijgave_Tourniquets_OK  ; Vrijgave Tourniquets OK Plc 1& Plc 2
ANDNOT 90.02
+(400) D_TOURN_L_TEL +1 D_TOURN_L_TEL  ; TEL AANTAL TOURNIKET LINKS
; rung 1: Splits drukknop tourniquets uit in : / Blokkeer tourniquet / Verhoog aantal
LD M_OS_VRIJGAVE_LINKSE_TOURNIQUET  ; Merker One Shot Vrijgave Linkse Tourniquet
OUT TR0
AND<(310) D_TOURN_L_TEL D_TOURN_L_MAX  ; TEL AANTAL TOURNIKET LINKS, MAX AANTAL TOURNIKET LINKS
OUT W90.00  ; Blokkeer Tourniquet
LD TR0
AND>=(325) D_TOURN_L_TEL D_TOURN_L_MAX  ; TEL AANTAL TOURNIKET LINKS, MAX AANTAL TOURNIKET LINKS
OUT W90.01  ; Verhoog aantal
; rung 2: Blokkeer tourniquet
LD P_On
OUT TR0
AND M_OS_OPEN_SLUIT_L_OEVER_POORTJES  ; Merker One Shot Open / Sluit Linker Poortjes Oever
ANDNOT 3327.01  ; Inganspoort links gesloten van PLC2
LD TR0
AND W90.00  ; Blokkeer Tourniquet
OUT TR1
ANDNOT W90.02  ; Blokkeer tourniquet links
ORLD
LD TR1
AND W90.02  ; Blokkeer tourniquet links
LD TR0
AND 3327.01  ; Inganspoort links gesloten van PLC2
@AND M_Show_Stap_1  ; Show Stap 1
ORLD
KEEP(011) W90.02  ; Blokkeer tourniquet links

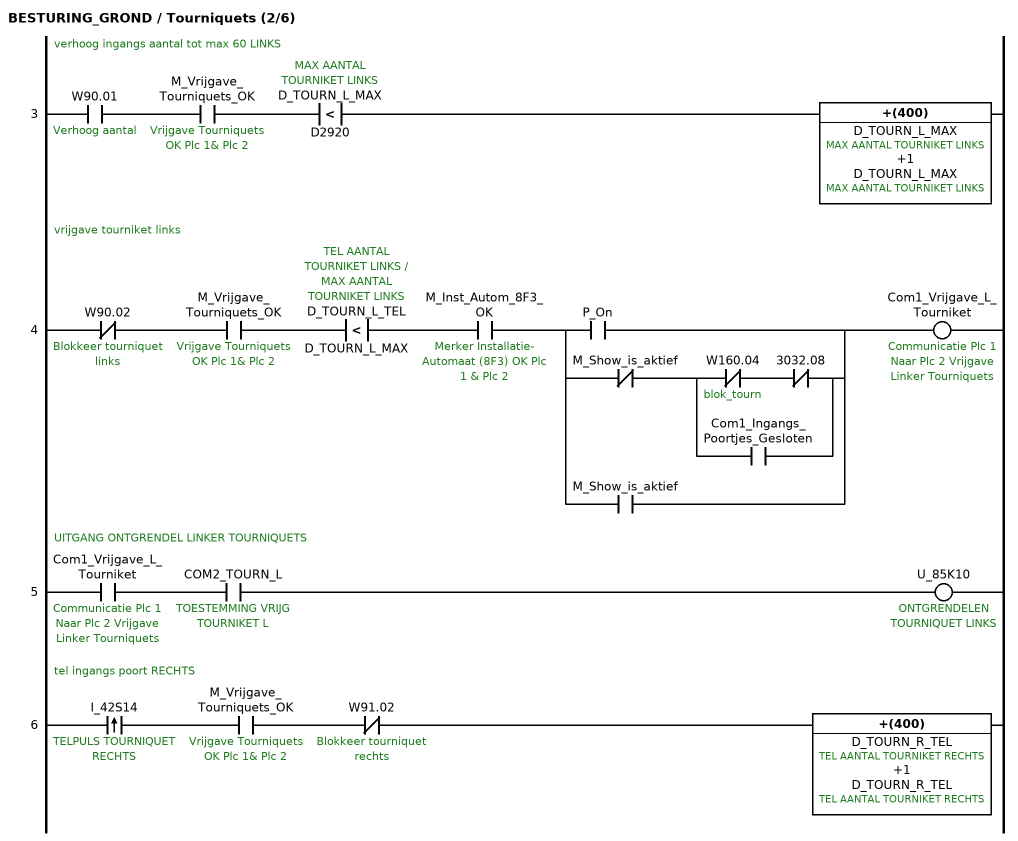
; rung 3: verhoog ingangs aantal tot max 60 LINKS
LD W90.01  ; Verhoog aantal
AND M_Vrijgave_Tourniquets_OK  ; Vrijgave Tourniquets OK Plc 1& Plc 2
AND<S(312) D_TOURN_L_MAX D2920  ; MAX AANTAL TOURNIKET LINKS
+(400) D_TOURN_L_MAX +1 D_TOURN_L_MAX  ; MAX AANTAL TOURNIKET LINKS
; rung 4: vrijgave tourniket links
LDNOT W90.02  ; Blokkeer tourniquet links
AND M_Vrijgave_Tourniquets_OK  ; Vrijgave Tourniquets OK Plc 1& Plc 2
AND<S(312) D_TOURN_L_TEL D_TOURN_L_MAX  ; TEL AANTAL TOURNIKET LINKS, MAX AANTAL TOURNIKET LINKS
AND M_Inst_Autom_8F3_OK  ; Merker Installatie-Automaat (8F3) OK Plc 1 & Plc 2
LD P_On
LDNOT M_Show_is_aktief
LDNOT W160.04  ; blok_tourn
ANDNOT 3032.08
OR Com1_Ingangs_Poortjes_Gesloten
ANDLD
ORLD
OR M_Show_is_aktief
ANDLD
OUT Com1_Vrijgave_L_Tourniket  ; Communicatie Plc 1 Naar Plc 2 Vrijgave Linker Tourniquets
; rung 5: UITGANG ONTGRENDEL LINKER TOURNIQUETS
LD Com1_Vrijgave_L_Tourniket  ; Communicatie Plc 1 Naar Plc 2 Vrijgave Linker Tourniquets
AND COM2_TOURN_L  ; TOESTEMMING VRIJG TOURNIKET L
OUT U_85K10  ; ONTGRENDELEN TOURNIQUET LINKS
; rung 6: tel ingangs poort RECHTS
@LD I_42S14  ; TELPULS TOURNIQUET RECHTS
AND M_Vrijgave_Tourniquets_OK  ; Vrijgave Tourniquets OK Plc 1& Plc 2
ANDNOT W91.02  ; Blokkeer tourniquet rechts
+(400) D_TOURN_R_TEL +1 D_TOURN_R_TEL  ; TEL AANTAL TOURNIKET RECHTS

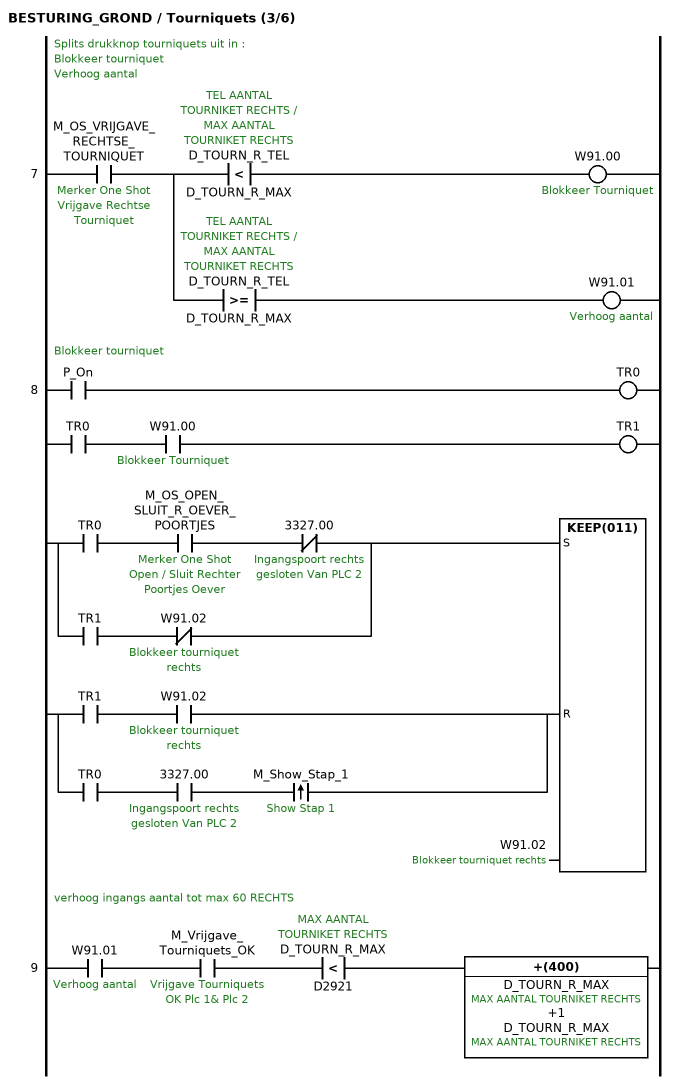
; rung 7: Splits drukknop tourniquets uit in : / Blokkeer tourniquet / Verhoog aantal
LD M_OS_VRIJGAVE_RECHTSE_TOURNIQUET  ; Merker One Shot Vrijgave Rechtse Tourniquet
OUT TR0
AND<(310) D_TOURN_R_TEL D_TOURN_R_MAX  ; TEL AANTAL TOURNIKET RECHTS, MAX AANTAL TOURNIKET RECHTS
OUT W91.00  ; Blokkeer Tourniquet
LD TR0
AND>=(325) D_TOURN_R_TEL D_TOURN_R_MAX  ; TEL AANTAL TOURNIKET RECHTS, MAX AANTAL TOURNIKET RECHTS
OUT W91.01  ; Verhoog aantal
; rung 8: Blokkeer tourniquet
LD P_On
OUT TR0
AND M_OS_OPEN_SLUIT_R_OEVER_POORTJES  ; Merker One Shot Open / Sluit Rechter Poortjes Oever
ANDNOT 3327.00  ; Ingangspoort rechts gesloten Van PLC 2
LD TR0
AND W91.00  ; Blokkeer Tourniquet
OUT TR1
ANDNOT W91.02  ; Blokkeer tourniquet rechts
ORLD
LD TR1
AND W91.02  ; Blokkeer tourniquet rechts
LD TR0
AND 3327.00  ; Ingangspoort rechts gesloten Van PLC 2
@AND M_Show_Stap_1  ; Show Stap 1
ORLD
KEEP(011) W91.02  ; Blokkeer tourniquet rechts
; rung 9: verhoog ingangs aantal tot max 60 RECHTS
LD W91.01  ; Verhoog aantal
AND M_Vrijgave_Tourniquets_OK  ; Vrijgave Tourniquets OK Plc 1& Plc 2
AND<S(312) D_TOURN_R_MAX D2921  ; MAX AANTAL TOURNIKET RECHTS
+(400) D_TOURN_R_MAX +1 D_TOURN_R_MAX  ; MAX AANTAL TOURNIKET RECHTS

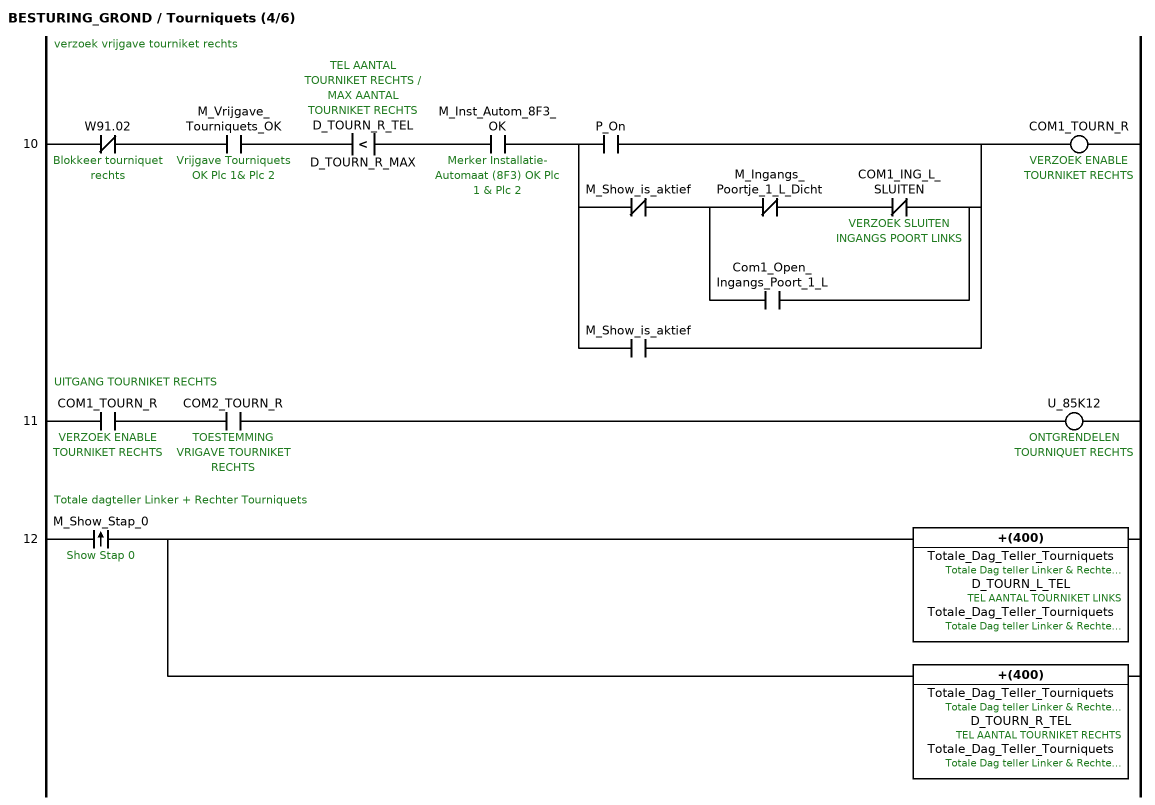
; rung 10: verzoek vrijgave tourniket rechts
LDNOT W91.02  ; Blokkeer tourniquet rechts
AND M_Vrijgave_Tourniquets_OK  ; Vrijgave Tourniquets OK Plc 1& Plc 2
AND<S(312) D_TOURN_R_TEL D_TOURN_R_MAX  ; TEL AANTAL TOURNIKET RECHTS, MAX AANTAL TOURNIKET RECHTS
AND M_Inst_Autom_8F3_OK  ; Merker Installatie-Automaat (8F3) OK Plc 1 & Plc 2
LD P_On
LDNOT M_Show_is_aktief
LDNOT M_Ingangs_Poortje_1_L_Dicht
ANDNOT COM1_ING_L_SLUITEN  ; VERZOEK SLUITEN INGANGS POORT LINKS
OR Com1_Open_Ingangs_Poort_1_L
ANDLD
ORLD
OR M_Show_is_aktief
ANDLD
OUT COM1_TOURN_R  ; VERZOEK ENABLE TOURNIKET RECHTS
; rung 11: UITGANG TOURNIKET RECHTS
LD COM1_TOURN_R  ; VERZOEK ENABLE TOURNIKET RECHTS
AND COM2_TOURN_R  ; TOESTEMMING VRIGAVE TOURNIKET RECHTS
OUT U_85K12  ; ONTGRENDELEN TOURNIQUET RECHTS
; rung 12: Totale dagteller Linker + Rechter Tourniquets
@LD M_Show_Stap_0  ; Show Stap 0
+(400) Totale_Dag_Teller_Tourniquets D_TOURN_L_TEL Totale_Dag_Teller_Tourniquets  ; Totale Dag teller Linker & Rechter Tournoquets, TEL AANTAL TOURNIKET LINKS
+(400) Totale_Dag_Teller_Tourniquets D_TOURN_R_TEL Totale_Dag_Teller_Tourniquets  ; Totale Dag teller Linker & Rechter Tournoquets, TEL AANTAL TOURNIKET RECHTS

